Staubli VAL3: insert_aOutput.pgx

public program insert_aOutput(string x_sItem (dimensions=1), bool x_bActive (dimensions=1), aio x_aDio (dimensions=1))
begin
  // insert a new IO
  if isDefined(aOutput[x_sItem])==false and ioStatus(x_aDio)>=0
    insert(aOutput[x_sItem])
    aOutput[x_sItem].bActive=x_bActive
    aOutput[x_sItem].sID=x_sItem
    aOutput[x_sItem].sName=x_sItem
    aioLink(aOutput[x_sItem].aAio,x_aDio)
    aOutput[x_sItem].bEnable=true
  endIf
end
